// TIA Portal V20 export
// export: Created 2025-12-01T14:56:22.0061297Z, ExportSetting None, DisplayName Totally Integrated Automation Portal, DisplayVersion V20 Update 3, DisplayName TIA Portal Openness, DisplayVersion V20 Update 3, DisplayName TIA Portal Version Control Interface, DisplayVersion V20 Update 3, DisplayName STEP 7 Professional, DisplayVersion V20 Update 3, DisplayName STEP 7 Safety, DisplayVersion V20 Update 2, DisplayName WinCC Basic/Comfort/Advanced, DisplayVersion V20 Update 3, DisplayName WinCC Professional, DisplayVersion V20 Update 3, DisplayName WinCC Unified, DisplayVersion V20 Update 3
TYPE "NDD_Enfardadora_Input"
   STRUCT
      BitDeVida : Bool;
      Libre_01 : Bool;
      Libre_02 : Bool;
      Libre_03 : Bool;
      Libre_04 : Bool;
      Libre_05 : Bool;
      Libre_06 : Bool;
      Libre_07 : Bool;
      AutoSinAnomalia : Bool;
      MarchaParo : Bool;
      Error : Bool;
      EnvolvedoraHomeReposo : Bool;
      EnvolvedoraEnMovimiento : Bool;
      ReameSeguridadULMA : Bool;
      EnvolvedoraSelectorAuto : Bool;   // Libre_16 (Antes)
      EnvolvedorapHs : Bool;   // AlturaPaleta (Antes)
      PeticionSubirElevador : Bool;
      PeticionBajarElevador : Bool;
      StopElevadorSoldar : Bool;
      Libre_23 : Bool;
      PermisoBajadaCapa : Bool;
      Libre_25 : Bool;
      EvacuarPaleta : Bool;
      CicloCompletado : Bool;
      Libre_30 : Bool;
      Libre_31 : Bool;
      Libre_32 : Bool;
      Libre_33 : Bool;
      Libre_34 : Bool;
      Libre_35 : Bool;
      AL_Rotura_Film : Bool;
      AL_Preaviso_Film : Bool;
      VelocidadElevador : Int;
      AlturaInicioEnfardado : Int;
      Libre_Int_08 : Int;
   END_STRUCT;
END_TYPE
